TYPE ST_EAPAxeState : 
	STRUCT
		(*   Actual Position mm  *)
		Position : LREAL := 0;
		(*   Actual Velocity  mm/s  *)
		Velocity : LREAL := 0;
		(*   Actual Torque   *)
		Torque : REAL := 0;
		(*   Error Code   *)
		Error : UDINT := 0;
		(*   TRUE=Power Enable   *)
		PowerActive : BOOL := false;
		(*  Home ok  *)
		Homed : BOOL := false;
	END_STRUCT
END_TYPE

(* stored: Version 1.1.0.1, ProductVersion 3.1.4024.11
   DUT ST_EAPAxeState: Id {b2bf15a3-216e-4778-bee0-f5139f667218} *)
